FUNCTION_BLOCK PusherControllerIReq (* Pusher Controller Interface Requier *)
  (* Standard: 61499-2 *)
  (* Version 0.2, 2003-12-05, JHC, Rockwell Automation, Renamed from NEWCOMPFB. *)
  (* Version 0.1, 2002-01-08, JHC, Rockwell Automation, Added DLY FB as example. *)
  (* Version 0.0, 2000-05-27, JHC, Rockwell Automation *)
  (* Compiler header: package fb.rt.dasdA1.A2.Pusher; *)
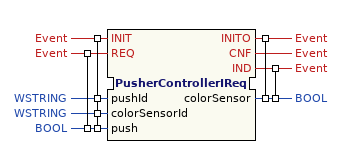
  EVENT_INPUT
    INIT WITH pushId, colorSensorId, push; (* Initialization Request *)
    REQ WITH push; (* Normal Execution Request *)
  END_EVENT
  EVENT_OUTPUT
    INITO WITH colorSensor; (* Initialization Confirm *)
    CNF; (* Execution Confirmation *)
    IND WITH colorSensor;
  END_EVENT
  VAR_INPUT
    pushId : WSTRING; (* Push event id *)
    colorSensorId : WSTRING; (* Id of the color sensor *)
    push : BOOL;
  END_VAR
  VAR_OUTPUT
    colorSensor : BOOL;
  END_VAR
  FBS
    pusherColorSensor : SUBL_1;
    pusherPush : PUBL_1;
  END_FBS
  EVENT_CONNECTIONS
    pusherColorSensor.INITO TO INITO;
    pusherColorSensor.IND TO CNF;
    INIT TO pusherPush.INIT;
    REQ TO pusherPush.REQ;
    pusherPush.INITO TO pusherColorSensor.INIT;
    pusherPush.CNF TO CNF;
    pusherColorSensor.IND TO IND;
  END_CONNECTIONS
  DATA_CONNECTIONS
    colorSensorId TO pusherColorSensor.ID;
    pusherColorSensor.RD_1 TO colorSensor;
    push TO pusherPush.SD_1;
    pushId TO pusherPush.ID;
  END_CONNECTIONS
END_FUNCTION_BLOCK
